TYPE ST_MESSAGE_CTRL :
STRUCT
  Cmd         : E_MESSAGE_CTRL;
END_STRUCT
END_TYPE

(* stored: Version 1.1.0.1, ProductVersion 3.1.4026.13
   DUT ST_MESSAGE_CTRL: Id {0947409c-e2ad-40e0-b722-4df7636e200a} *)
